PROGRAM prgCalc
VAR
	//Sum of all CEE32 Measurements
	fbEMTotalCounter		: FB_EnergyCounter;
	lr_RealPower_Total		: LREAL;					//{#lynus.ag#()}
END_VAR

VAR PERSISTENT
	lr_EnergyCounter_Total	: LREAL;					//{#lynus.ag#()}
END_VAR


lr_RealPower_Total := 	prgEM.lr_RealPower_EM1 + 
						prgEM.lr_RealPower_EM2 + 
						prgEM.lr_RealPower_EM3 + 
						prgEM.lr_RealPower_EM4 + 
						prgEM.lr_RealPower_EM5 + 
						prgEM.lr_RealPower_EM6 + 
						prgEM.lr_RealPower_EM7 + 
						prgEM.lr_RealPower_EM8 + 
						prgEM.lr_RealPower_EM9;

fbEMTotalCounter(
	byActiveTariff:= 1, 
	lrPowerInput:= lr_RealPower_Total, 
	lrTotalCounterEnergy_Consumption=> , 
	lrTotalCounterEnergy_Production=> , 
	lrCounterEnergyT1_Consumption=> , 
	lrCounterEnergyT2_Consumption=> , 
	lrCounterEnergyT1_Production=> , 
	lrCounterEnergyT2_Production=> );
	
IF fbEMTotalCounter.lrTotalCounterEnergy_Consumption > lr_EnergyCounter_Total THEN  	
	lr_EnergyCounter_Total := fbEMTotalCounter.lrTotalCounterEnergy_Consumption;
END_IF

END_PROGRAM

(* stored: Version 1.1.0.1, ProductVersion 3.1.4024.12
   POU prgCalc: Id {323b95c0-48b6-42d5-83da-8e9a5d861f73}, SpecialFunc None *)
